TYPE incCommSettings :
STRUCT
END_STRUCT
END_TYPE

(* stored: Version 1.1.0.1, ProductVersion 3.1.4024.3
   DUT incCommSettings: Id {f5fee06c-c2fa-41ea-811b-7b814e26fd20} *)
